(* PLC project Modbus_Test_Project_Abingdon_Virtual.project, CODESYS CODESYS V3.5 SP20 Patch 5 *)
(* stored: creationDateTime 2025-07-04T16:22:35.3439176, modificationDateTime 2025-07-04T16:22:08.6346008 *)

TYPE StructModbusDataforTCPServer : STRUCT
  aReadCoils : ARRAY[1..100] OF BYTE;
  aWriteCoils : ARRAY[1..100] OF BYTE;
  aReadDiscreteInputs : ARRAY[1..100] OF BYTE;
  aWriteDiscreteInputs : ARRAY[1..100] OF BYTE;
  aReadHoldingRegisters : ARRAY[1..100] OF INT;
  aWriteHoldingRegisters : ARRAY[1..100] OF INT;
  aReadInputRegisters : ARRAY[1..100] OF INT;
  aWriteInputRegisters : ARRAY[1..100] OF INT;
END_STRUCT;
END_TYPE

PROGRAM Main
  VAR
    nCounter : INT;
    bInit : BOOL := FALSE;
    ModbusTcpServer : CmpModbusTcpServer.ModbusServer;  (* Modbus Tcp Server *)
    ModbusTcpServerDevice : CmpModbusTcpServer.ModbusServerDevice;
    stModbusTcpServerData : StructModbusDataForTCPServer;
    stModbusTcpServerStatus : CmpModbusTcpServer.Status;
    strModataData : StructModbusDataforTCPServer;
  END_VAR

                    nCounter := nCounter + 1;

IF bInit = FALSE THEN
	bInit := TRUE;
	ModbusTcpServerDevice.Initialize(usiUnitId := 1);

	ModbusTcpServer.Initialize(
		pbyIpAddress:=ADR('192.168.3.102'), 
		uiPort:= 1100);

	ModbusTcpServer.Open();
END_IF

ModbusTcpServerDevice.ReadCoils(
	uiStartAddress:=0,
	uiReadLength:=10,
	pbyBuffer:= ADR(strModataData.aReadCoils), 
	uiBufferSize:=10);

ModbusTcpServerDevice.WriteCoils(
	uiStartAddress:=100,
	uiWriteLength:=10,
	pbyBuffer:= ADR(strModataData.aWriteCoils), 
	uiBufferSize:=10);

ModbusTcpServerDevice.ReadDiscreteInputs(
	uiStartAddress:=0,
	uiReadLength:=10, 
	pbyBuffer:= ADR(strModataData.aReadDiscreteInputs), 
	uiBufferSize:=10);

ModbusTcpServerDevice.WriteDiscreteInputs(
	uiStartAddress:=100,
	uiWriteLength:=10,
	pbyBuffer:= ADR(strModataData.aWriteDiscreteInputs), 
	uiBufferSize:=10);

ModbusTcpServerDevice.ReadHoldingRegisters(
	uiStartAddress:=0, 
	uiReadLength:=10, 
	pwBuffer:= ADR(strModataData.aReadHoldingRegisters), 
	uiBufferSize:=20);
	
ModbusTcpServerDevice.WriteHoldingRegisters(
	uiStartAddress:=100, 
	uiWriteLength:=10,
	pwBuffer:= ADR(strModataData.aWriteHoldingRegisters), 
	uiBufferSize:=20);

ModbusTcpServerDevice.ReadInputRegisters(
	uiStartAddress:=0, 
	uiReadLength:=10,
	pwBuffer:= ADR(strModataData.aReadInputRegisters), 
	uiBufferSize:=20);

ModbusTcpServerDevice.WriteInputRegisters(
	uiStartAddress:=100, 
	uiWriteLength:=10,
	pwBuffer:= ADR(strModataData.aWriteInputRegisters), 
	uiBufferSize:=20);

ModbusTcpServer.GetStatus(
	pStatus:=ADR(stModbusTcpServerStatus));
                  
END_PROGRAM

CONFIGURATION EDWARDS_ARM_Cortex
  RESOURCE Application ON PLC
    TASK Task(INTERVAL := T#100ms, PRIORITY := 1);
    PROGRAM Main WITH Task : Main;
  END_RESOURCE
END_CONFIGURATION
